(* Logix 5000 project; controller Tetris Emulate 5570 rev 35.11; software revision 35.00 *)

TASK MainTask (continuous, watchdog 500 ms) : MainProgram

MODULES
   Local : Emulate 5570 (ICP 2, rev 35.11)
END_MODULES

VAR_GLOBAL   (* controller tags *)
   AVE_Control : CONTROL := (LEN := 3);
   AVE_Dest : DINT;
   Background_Color_Matrix : SINT[12,8] := ([5,3] := 3, [6,3] := 3, [7,3] := 3, [8,3] := 3);
   Background_Matrix : SINT[12,8] := ([5,3] := 1, [6,3] := 1, [7,3] := 1, [8,3] := 1, [10,4] := 1, [10,5] := 1, [10,6] := 1, [10,7] := 1, [11,4] := 1, [11,5] := 1, [11,6] := 1, [11,7] := 1);
   Background_Saved_Color_Matrix : SINT[12,8];
   Clear_Color_Matrix : SINT[12,8];
   Clear_Matrix : SINT[12,8] := ([10,4] := 1, [10,5] := 1, [10,6] := 1, [10,7] := 1, [11,4] := 1, [11,5] := 1, [11,6] := 1, [11,7] := 1);
   Clear_Row_For_Index : DINT;
   Clock_Enable : BOOL := 1;
   CTU_Clock : COUNTER := (PRE := 2, ACC := 3, DN := 1);
   CTU_Clock_Reset : COUNTER := (PRE := 4, ACC := 3);
   Current_Piece_X_Size : DINT := 1;
   Current_Piece_Y_Size : DINT := 4;
   Current_X : SINT := 3;
   Current_Y : SINT := 5;
   Current_Y_Limit : DINT := 8;
   GSV_DateTime : DINT[7] := ([0] := 2025, [1] := 6, [2] := 5, [3] := 22, [4] := 27, [5] := 29, [6] := 833012);
   Input_Piece : SINT := 4;
   Master_Clear : BOOL;
   Next_Row_Check : SINT[8];
   ONS_Clock : BOOL := 1;
   ONS_Left : BOOL;
   ONS_Piece_Stopped : BOOL := 1;
   ONS_Right : BOOL;
   ONS_Rotate : BOOL;
   ONS_Score : BOOL[32];
   Piece_1_Matrix_R0 : SINT[2,3] := ([0,1] := 1, [1,0] := 1, [1,1] := 1, [1,2] := 1);
   Piece_1_Matrix_R1 : SINT[3,2] := ([0,0] := 1, [1,0] := 1, [1,1] := 1, [2,0] := 1);
   Piece_1_Matrix_R2 : SINT[2,3] := ([0,0] := 1, [0,1] := 1, [0,2] := 1, [1,1] := 1);
   Piece_1_Matrix_R3 : SINT[3,2] := ([0,1] := 1, [1,0] := 1, [1,1] := 1, [2,1] := 1);
   Piece_1_X : DINT;
   Piece_1_Y : INT;
   Piece_2_Matrix : SINT[2,2] := ([0,0] := 1, [0,1] := 1, [1,0] := 1, [1,1] := 1);
   Piece_3_Matrix_R0 : SINT[2,3] := ([0,0] := 1, [0,1] := 1, [1,1] := 1, [1,2] := 1);
   Piece_3_Matrix_R1 : SINT[3,2] := ([0,0] := 1, [1,0] := 1, [1,1] := 1, [2,1] := 1);
   Piece_4_Matrix_R0 : SINT[4,1] := ([0,0] := 1, [1,0] := 1, [2,0] := 1, [3,0] := 1);
   Piece_4_Matrix_R1 : SINT[1,4] := ([0,0] := 1, [0,1] := 1, [0,2] := 1, [0,3] := 1);
   Piece_Color : DINT := 3;
   Piece_Mov_Left : BOOL;
   Piece_Mov_Right : BOOL;
   Piece_Rotate : BOOL;
   Piece_Rotation : DINT;
   Piece_Type : SINT := 4;
   Previous_Color : DINT;
   Previous_Color_2 : DINT;
   Pulse_MS : BOOL;
   Reset : BOOL := 1;
   Saved_Matrix : SINT[12,8] := ([10,4] := 1, [10,5] := 1, [10,6] := 1, [10,7] := 1, [11,4] := 1, [11,5] := 1, [11,6] := 1, [11,7] := 1);
   Score : DINT;
   Start : BOOL;
   Update_Grid : BOOL;
END_VAR

PROGRAM MainProgram   (* main routine MainRoutine *)

ROUTINE Background_Clear   (* ladder *)
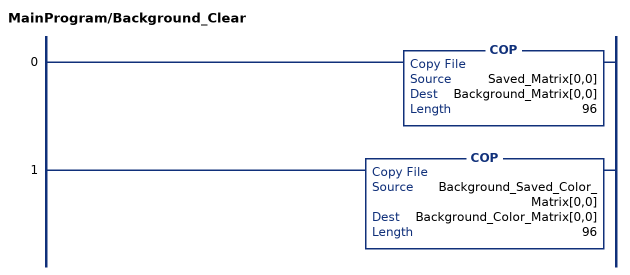
   0: COP(Saved_Matrix[0,0],Background_Matrix[0,0],96);
   1: COP(Background_Saved_Color_Matrix[0,0],Background_Color_Matrix[0,0],96);
END_ROUTINE

ROUTINE Clear_Full_Row   (* ladder *)
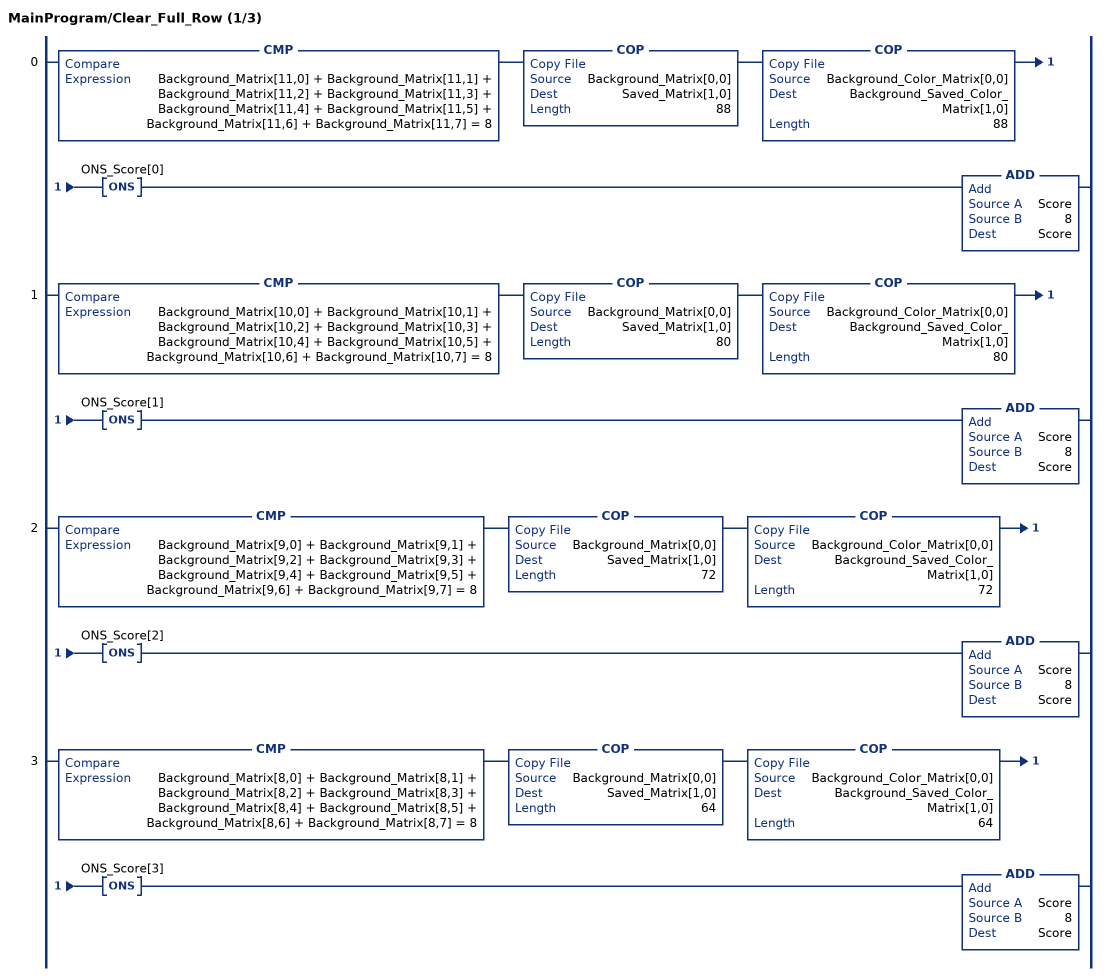
   0: CMP(Background_Matrix[11,0] + Background_Matrix[11,1] + Background_Matrix[11,2] + Background_Matrix[11,3] + Background_Matrix[11,4] + Background_Matrix[11,5] + Background_Matrix[11,6] + Background_Matrix[11,7] = 8)COP(Background_Matrix[0,0],Saved_Matrix[1,0],88)COP(Background_Color_Matrix[0,0],Background_Saved_Color_Matrix[1,0],88)ONS(ONS_Score[0])ADD(Score,8,Score);
   1: CMP(Background_Matrix[10,0] + Background_Matrix[10,1] + Background_Matrix[10,2] + Background_Matrix[10,3] + Background_Matrix[10,4] + Background_Matrix[10,5] + Background_Matrix[10,6] + Background_Matrix[10,7] = 8)COP(Background_Matrix[0,0],Saved_Matrix[1,0],80)COP(Background_Color_Matrix[0,0],Background_Saved_Color_Matrix[1,0],80)ONS(ONS_Score[1])ADD(Score,8,Score);
   2: CMP(Background_Matrix[9,0] + Background_Matrix[9,1] + Background_Matrix[9,2] + Background_Matrix[9,3] + Background_Matrix[9,4] + Background_Matrix[9,5] + Background_Matrix[9,6] + Background_Matrix[9,7] = 8)COP(Background_Matrix[0,0],Saved_Matrix[1,0],72)COP(Background_Color_Matrix[0,0],Background_Saved_Color_Matrix[1,0],72)ONS(ONS_Score[2])ADD(Score,8,Score);
   3: CMP(Background_Matrix[8,0] + Background_Matrix[8,1] + Background_Matrix[8,2] + Background_Matrix[8,3] + Background_Matrix[8,4] + Background_Matrix[8,5] + Background_Matrix[8,6] + Background_Matrix[8,7] = 8)COP(Background_Matrix[0,0],Saved_Matrix[1,0],64)COP(Background_Color_Matrix[0,0],Background_Saved_Color_Matrix[1,0],64)ONS(ONS_Score[3])ADD(Score,8,Score);
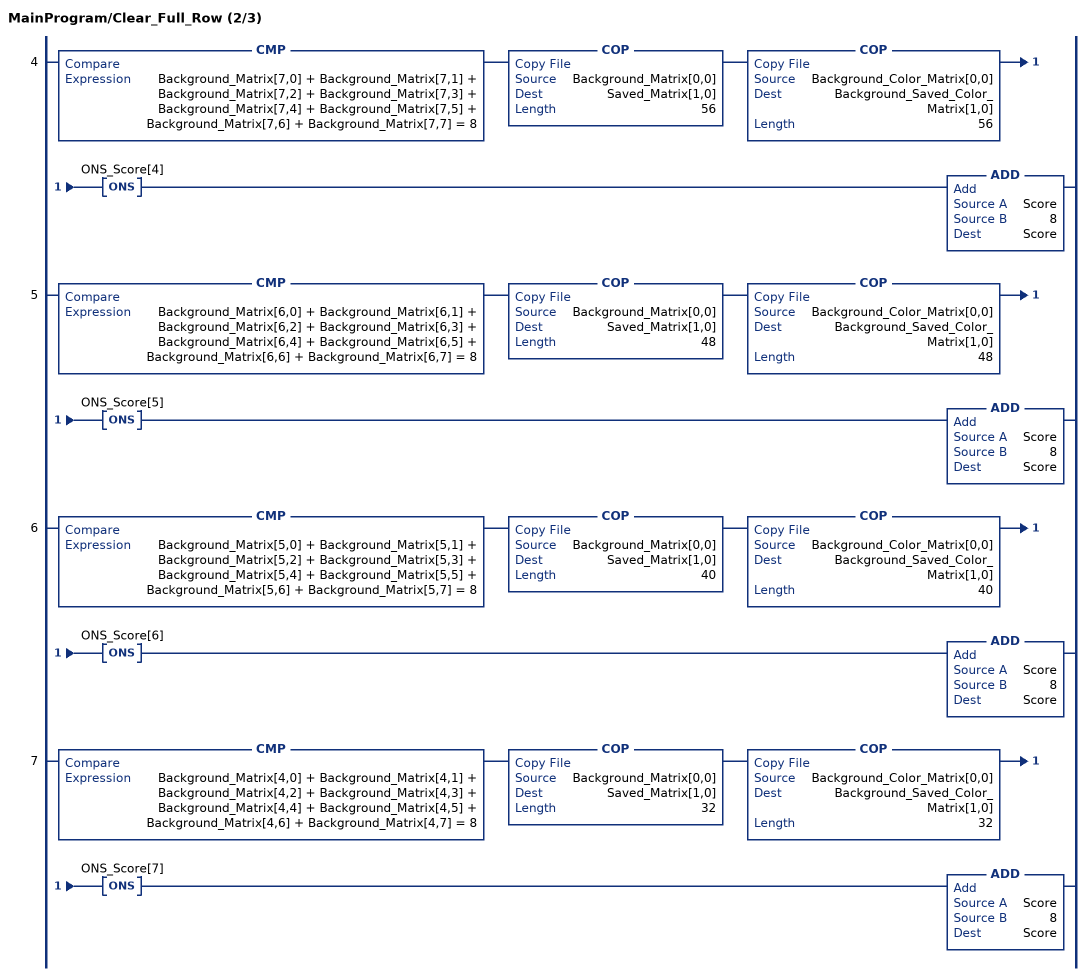
   4: CMP(Background_Matrix[7,0] + Background_Matrix[7,1] + Background_Matrix[7,2] + Background_Matrix[7,3] + Background_Matrix[7,4] + Background_Matrix[7,5] + Background_Matrix[7,6] + Background_Matrix[7,7] = 8)COP(Background_Matrix[0,0],Saved_Matrix[1,0],56)COP(Background_Color_Matrix[0,0],Background_Saved_Color_Matrix[1,0],56)ONS(ONS_Score[4])ADD(Score,8,Score);
   5: CMP(Background_Matrix[6,0] + Background_Matrix[6,1] + Background_Matrix[6,2] + Background_Matrix[6,3] + Background_Matrix[6,4] + Background_Matrix[6,5] + Background_Matrix[6,6] + Background_Matrix[6,7] = 8)COP(Background_Matrix[0,0],Saved_Matrix[1,0],48)COP(Background_Color_Matrix[0,0],Background_Saved_Color_Matrix[1,0],48)ONS(ONS_Score[5])ADD(Score,8,Score);
   6: CMP(Background_Matrix[5,0] + Background_Matrix[5,1] + Background_Matrix[5,2] + Background_Matrix[5,3] + Background_Matrix[5,4] + Background_Matrix[5,5] + Background_Matrix[5,6] + Background_Matrix[5,7] = 8)COP(Background_Matrix[0,0],Saved_Matrix[1,0],40)COP(Background_Color_Matrix[0,0],Background_Saved_Color_Matrix[1,0],40)ONS(ONS_Score[6])ADD(Score,8,Score);
   7: CMP(Background_Matrix[4,0] + Background_Matrix[4,1] + Background_Matrix[4,2] + Background_Matrix[4,3] + Background_Matrix[4,4] + Background_Matrix[4,5] + Background_Matrix[4,6] + Background_Matrix[4,7] = 8)COP(Background_Matrix[0,0],Saved_Matrix[1,0],32)COP(Background_Color_Matrix[0,0],Background_Saved_Color_Matrix[1,0],32)ONS(ONS_Score[7])ADD(Score,8,Score);
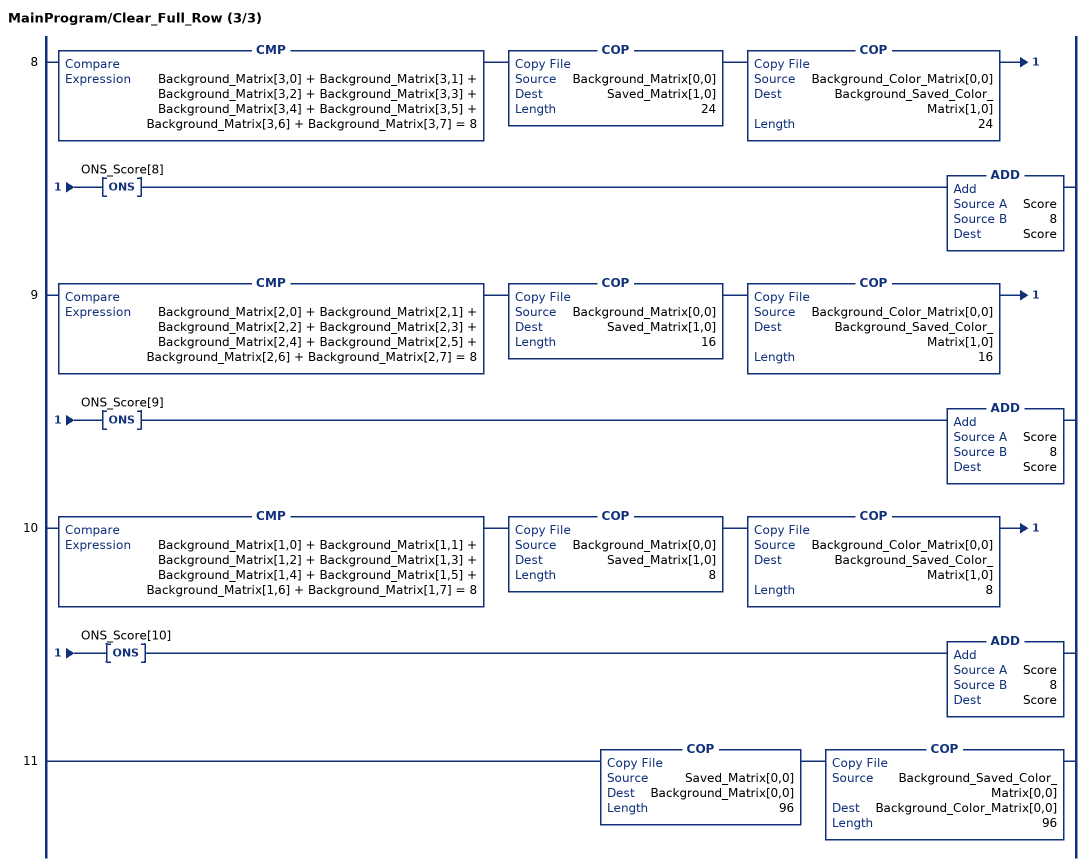
   8: CMP(Background_Matrix[3,0] + Background_Matrix[3,1] + Background_Matrix[3,2] + Background_Matrix[3,3] + Background_Matrix[3,4] + Background_Matrix[3,5] + Background_Matrix[3,6] + Background_Matrix[3,7] = 8)COP(Background_Matrix[0,0],Saved_Matrix[1,0],24)COP(Background_Color_Matrix[0,0],Background_Saved_Color_Matrix[1,0],24)ONS(ONS_Score[8])ADD(Score,8,Score);
   9: CMP(Background_Matrix[2,0] + Background_Matrix[2,1] + Background_Matrix[2,2] + Background_Matrix[2,3] + Background_Matrix[2,4] + Background_Matrix[2,5] + Background_Matrix[2,6] + Background_Matrix[2,7] = 8)COP(Background_Matrix[0,0],Saved_Matrix[1,0],16)COP(Background_Color_Matrix[0,0],Background_Saved_Color_Matrix[1,0],16)ONS(ONS_Score[9])ADD(Score,8,Score);
   10: CMP(Background_Matrix[1,0] + Background_Matrix[1,1] + Background_Matrix[1,2] + Background_Matrix[1,3] + Background_Matrix[1,4] + Background_Matrix[1,5] + Background_Matrix[1,6] + Background_Matrix[1,7] = 8)COP(Background_Matrix[0,0],Saved_Matrix[1,0],8)COP(Background_Color_Matrix[0,0],Background_Saved_Color_Matrix[1,0],8)ONS(ONS_Score[10])ADD(Score,8,Score);
   11: COP(Saved_Matrix[0,0],Background_Matrix[0,0],96)COP(Background_Saved_Color_Matrix[0,0],Background_Color_Matrix[0,0],96);
END_ROUTINE

ROUTINE Clock   (* ladder *)
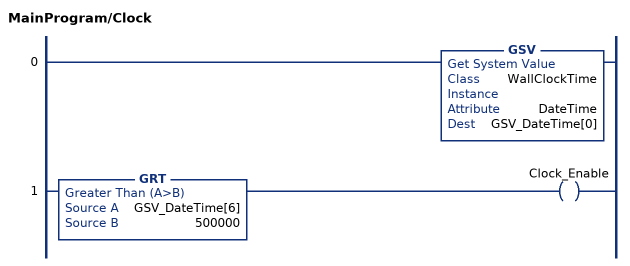
   0: GSV(WallClockTime,,DateTime,GSV_DateTime[0]);
   1: GRT(GSV_DateTime[6],500000)OTE(Clock_Enable);
END_ROUTINE

ROUTINE MainRoutine   (* ladder *)
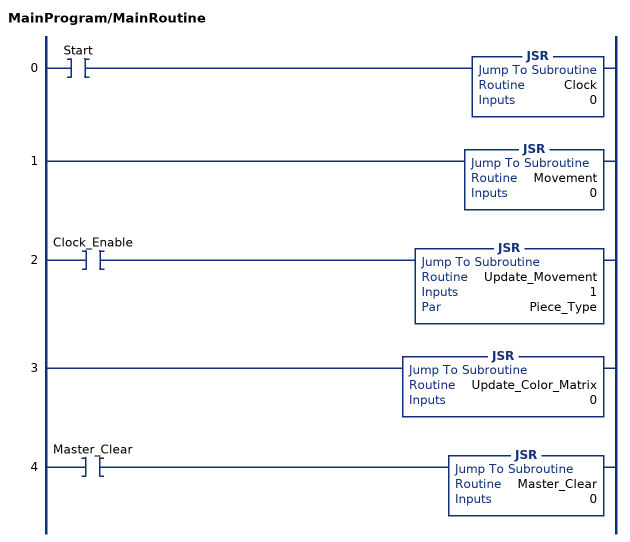
   0: XIC(Start)JSR(Clock,0);
   1: JSR(Movement,0);
   2: XIC(Clock_Enable)JSR(Update_Movement,1,Piece_Type);
   3: JSR(Update_Color_Matrix,0);
   4: XIC(Master_Clear)JSR(Master_Clear,0);
END_ROUTINE

ROUTINE Master_Clear   (* ladder *)
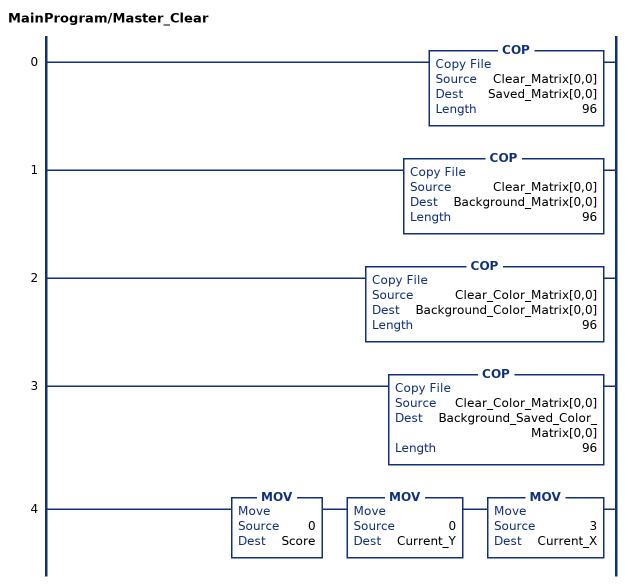
   0: COP(Clear_Matrix[0,0],Saved_Matrix[0,0],96);
   1: COP(Clear_Matrix[0,0],Background_Matrix[0,0],96);
   2: COP(Clear_Color_Matrix[0,0],Background_Color_Matrix[0,0],96);
   3: COP(Clear_Color_Matrix[0,0],Background_Saved_Color_Matrix[0,0],96);
   4: MOV(0,Score)MOV(0,Current_Y)MOV(3,Current_X);
END_ROUTINE

ROUTINE Movement   (* ladder *)
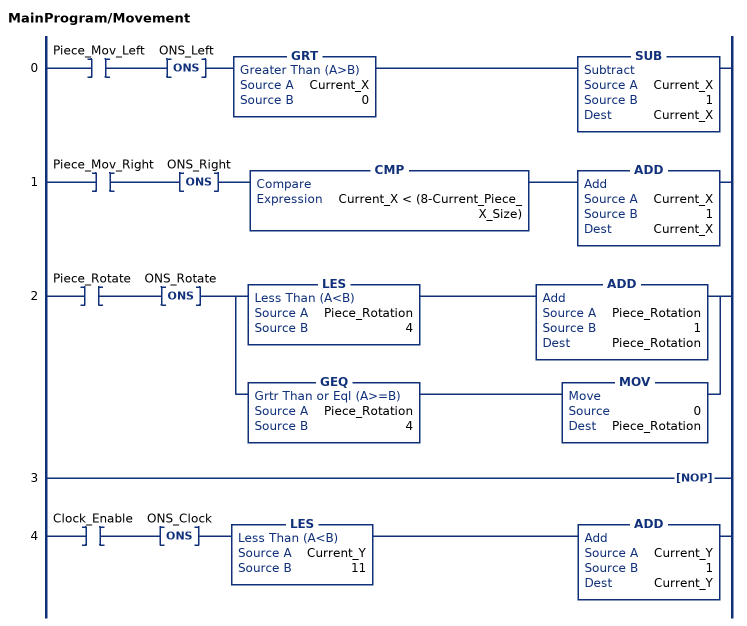
   0: XIC(Piece_Mov_Left)ONS(ONS_Left)GRT(Current_X,0)SUB(Current_X,1,Current_X);
   1: XIC(Piece_Mov_Right)ONS(ONS_Right)CMP(Current_X < (8-Current_Piece_X_Size))ADD(Current_X,1,Current_X);
   2: XIC(Piece_Rotate)ONS(ONS_Rotate)[LES(Piece_Rotation,4) ADD(Piece_Rotation,1,Piece_Rotation) ,GEQ(Piece_Rotation,4) MOV(0,Piece_Rotation) ];
   3: NOP();
   4: XIC(Clock_Enable)ONS(ONS_Clock)LES(Current_Y,11)ADD(Current_Y,1,Current_Y);
END_ROUTINE

ROUTINE Piece_1_Rotation   (* ladder *)
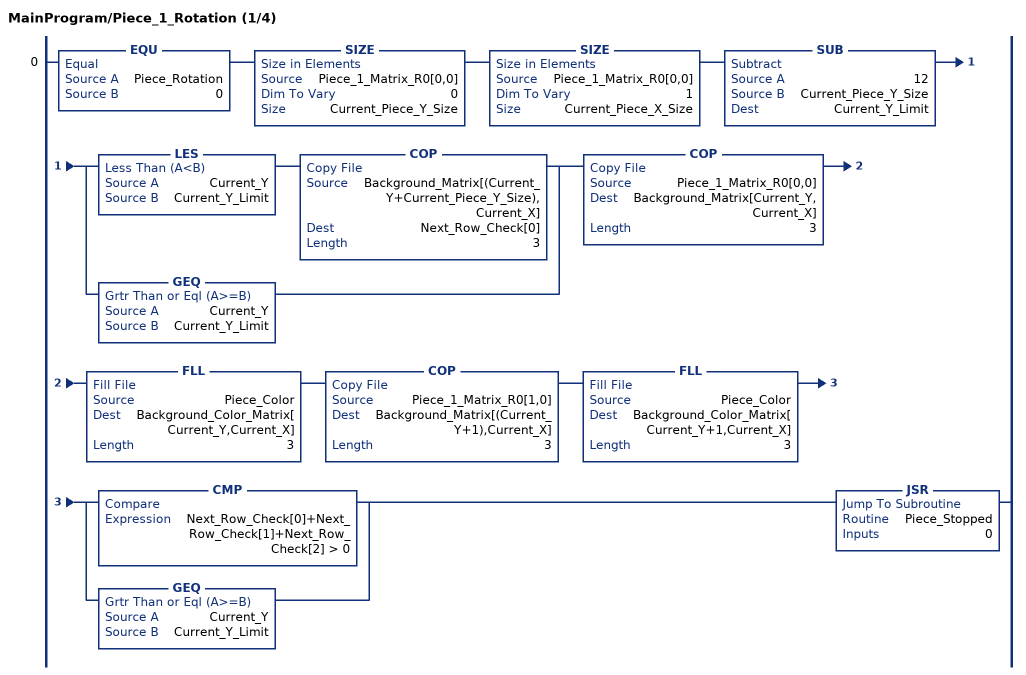
   0: EQU(Piece_Rotation,0)SIZE(Piece_1_Matrix_R0[0,0],0,Current_Piece_Y_Size)SIZE(Piece_1_Matrix_R0[0,0],1,Current_Piece_X_Size)SUB(12,Current_Piece_Y_Size,Current_Y_Limit)[LES(Current_Y,Current_Y_Limit) COP(Background_Matrix[(Current_Y+Current_Piece_Y_Size),Current_X],Next_Row_Check[0],3) ,GEQ(Current_Y,Current_Y_Limit) ]COP(Piece_1_Matrix_R0[0,0],Background_Matrix[Current_Y,Current_X],3)FLL(Piece_Color,Background_Color_Matrix[Current_Y,Current_X],3)COP(Piece_1_Matrix_R0[1,0],Background_Matrix[(Current_Y+1),Current_X],3)FLL(Piece_Color,Background_Color_Matrix[Current_Y+1,Current_X],3)[CMP(Next_Row_Check[0]+Next_Row_Check[1]+Next_Row_Check[2] > 0) ,GEQ(Current_Y,Current_Y_Limit) ]JSR(Piece_Stopped,0);
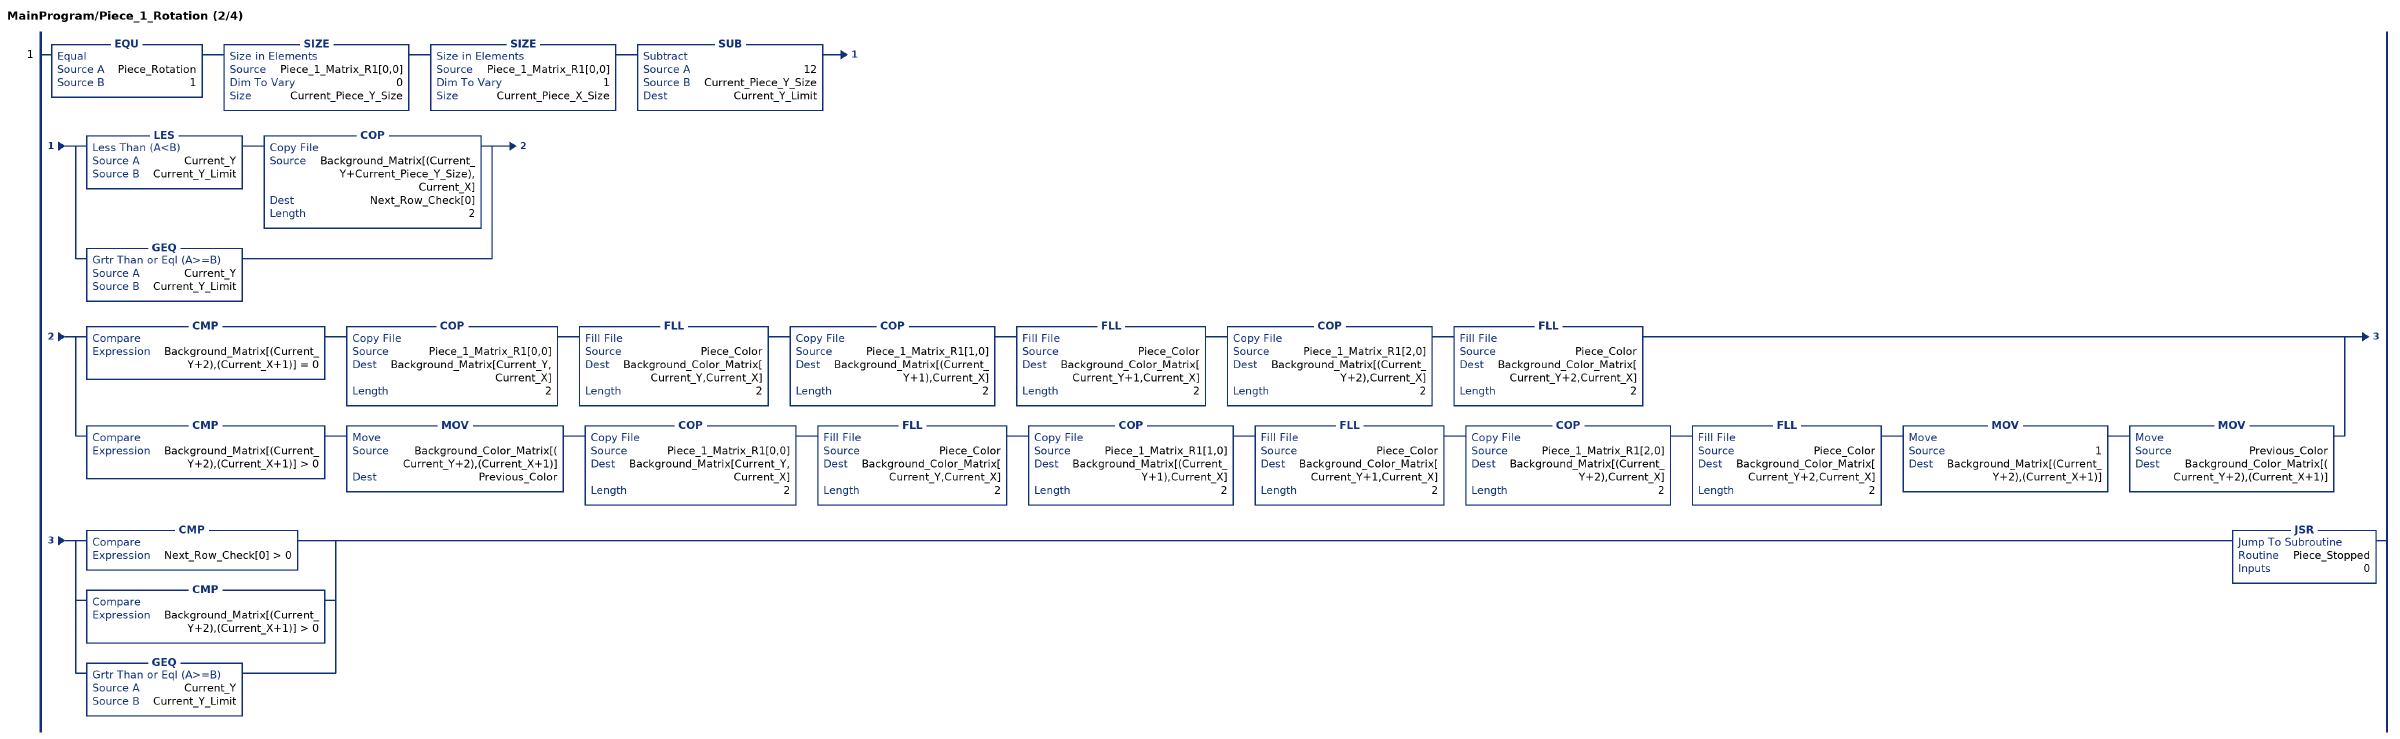
   1: EQU(Piece_Rotation,1)SIZE(Piece_1_Matrix_R1[0,0],0,Current_Piece_Y_Size)SIZE(Piece_1_Matrix_R1[0,0],1,Current_Piece_X_Size)SUB(12,Current_Piece_Y_Size,Current_Y_Limit)[LES(Current_Y,Current_Y_Limit) COP(Background_Matrix[(Current_Y+Current_Piece_Y_Size),Current_X],Next_Row_Check[0],2) ,GEQ(Current_Y,Current_Y_Limit) ][CMP(Background_Matrix[(Current_Y+2),(Current_X+1)] = 0) COP(Piece_1_Matrix_R1[0,0],Background_Matrix[Current_Y,Current_X],2) FLL(Piece_Color,Background_Color_Matrix[Current_Y,Current_X],2) COP(Piece_1_Matrix_R1[1,0],Background_Matrix[(Current_Y+1),Current_X],2) FLL(Piece_Color,Background_Color_Matrix[Current_Y+1,Current_X],2) COP(Piece_1_Matrix_R1[2,0],Background_Matrix[(Current_Y+2),Current_X],2) FLL(Piece_Color,Background_Color_Matrix[Current_Y+2,Current_X],2) ,CMP(Background_Matrix[(Current_Y+2),(Current_X+1)] > 0) MOV(Background_Color_Matrix[(Current_Y+2),(Current_X+1)],Previous_Color) COP(Piece_1_Matrix_R1[0,0],Background_Matrix[Current_Y,Current_X],2) FLL(Piece_Color,Background_Color_Matrix[Current_Y,Current_X],2) COP(Piece_1_Matrix_R1[1,0],Background_Matrix[(Current_Y+1),Current_X],2) FLL(Piece_Color,Background_Color_Matrix[Current_Y+1,Current_X],2) COP(Piece_1_Matrix_R1[2,0],Background_Matrix[(Current_Y+2),Current_X],2) FLL(Piece_Color,Background_Color_Matrix[Current_Y+2,Current_X],2) MOV(1,Background_Matrix[(Current_Y+2),(Current_X+1)]) MOV(Previous_Color,Background_Color_Matrix[(Current_Y+2),(Current_X+1)]) ][CMP(Next_Row_Check[0] > 0) ,CMP(Background_Matrix[(Current_Y+2),(Current_X+1)] > 0) ,GEQ(Current_Y,Current_Y_Limit) ]JSR(Piece_Stopped,0);
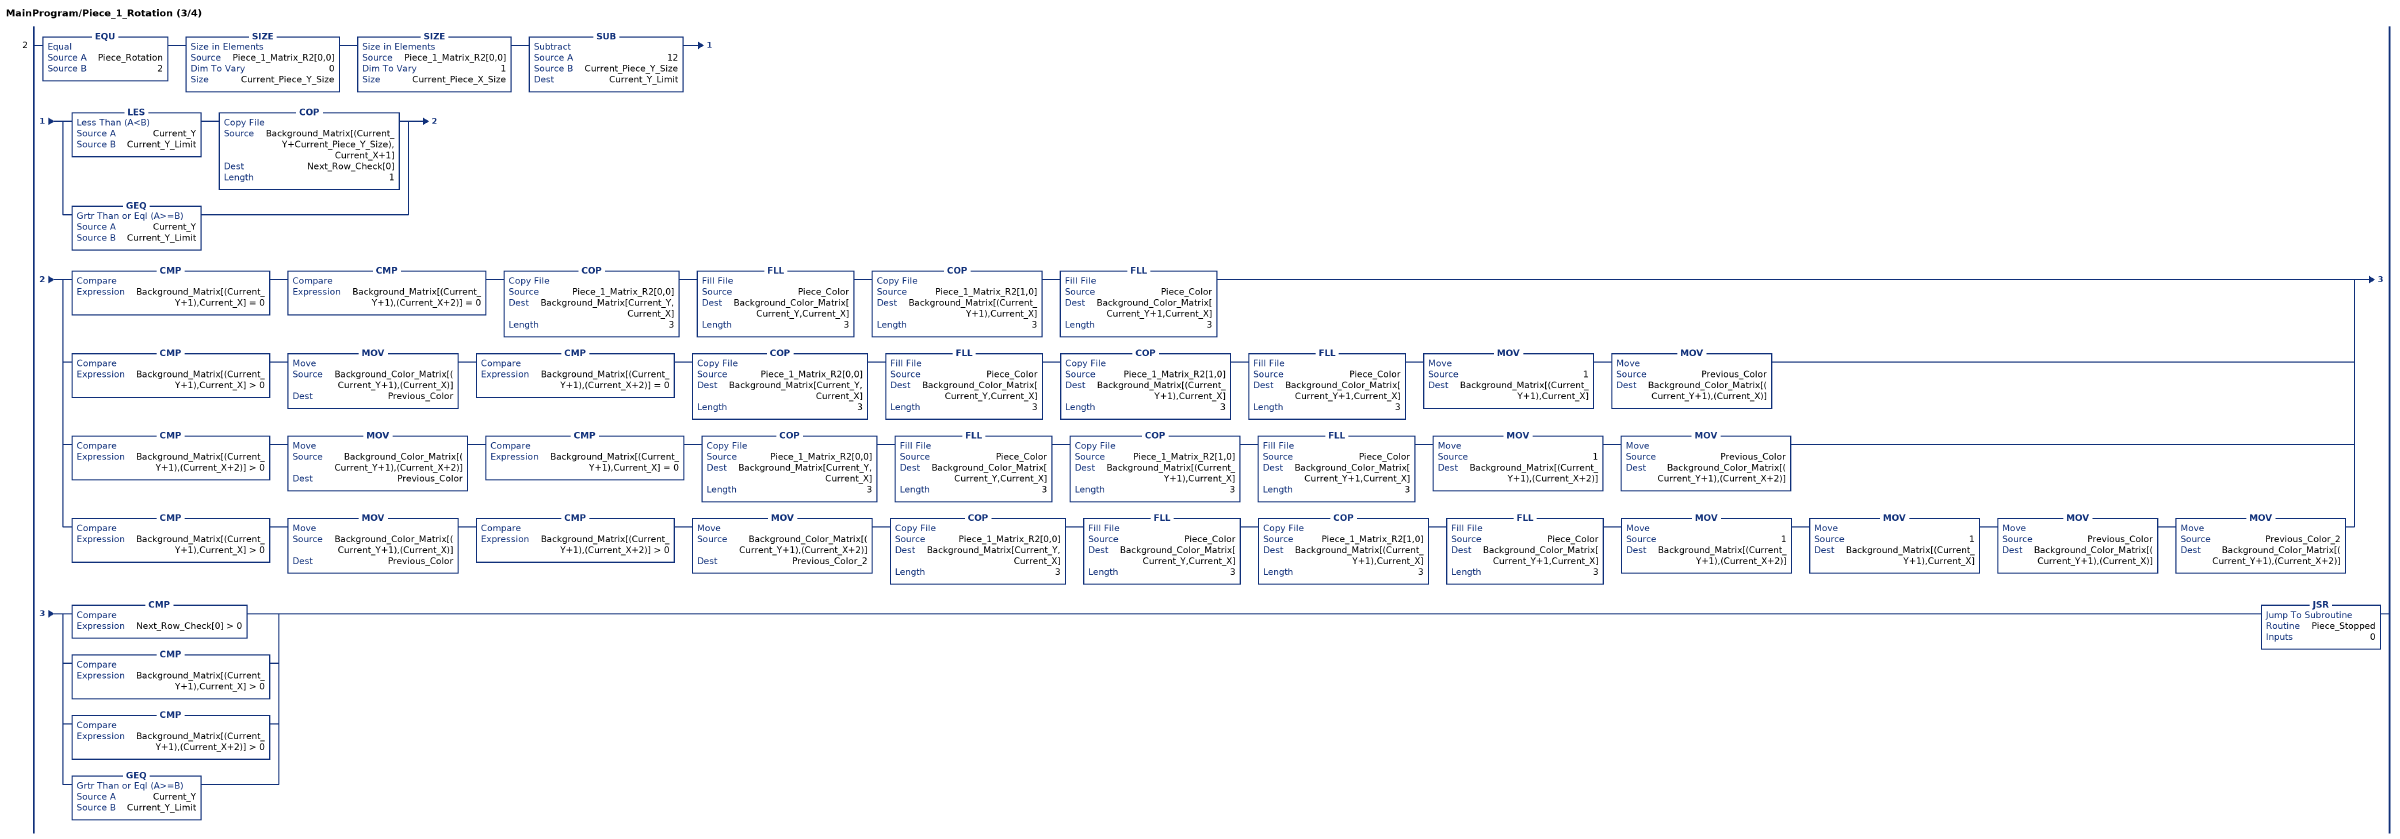
   2: EQU(Piece_Rotation,2)SIZE(Piece_1_Matrix_R2[0,0],0,Current_Piece_Y_Size)SIZE(Piece_1_Matrix_R2[0,0],1,Current_Piece_X_Size)SUB(12,Current_Piece_Y_Size,Current_Y_Limit)[LES(Current_Y,Current_Y_Limit) COP(Background_Matrix[(Current_Y+Current_Piece_Y_Size),Current_X+1],Next_Row_Check[0],1) ,GEQ(Current_Y,Current_Y_Limit) ][CMP(Background_Matrix[(Current_Y+1),Current_X] = 0) CMP(Background_Matrix[(Current_Y+1),(Current_X+2)] = 0) COP(Piece_1_Matrix_R2[0,0],Background_Matrix[Current_Y,Current_X],3) FLL(Piece_Color,Background_Color_Matrix[Current_Y,Current_X],3) COP(Piece_1_Matrix_R2[1,0],Background_Matrix[(Current_Y+1),Current_X],3) FLL(Piece_Color,Background_Color_Matrix[Current_Y+1,Current_X],3) ,[CMP(Background_Matrix[(Current_Y+1),Current_X] > 0) MOV(Background_Color_Matrix[(Current_Y+1),(Current_X)],Previous_Color) CMP(Background_Matrix[(Current_Y+1),(Current_X+2)] = 0) COP(Piece_1_Matrix_R2[0,0],Background_Matrix[Current_Y,Current_X],3) FLL(Piece_Color,Background_Color_Matrix[Current_Y,Current_X],3) COP(Piece_1_Matrix_R2[1,0],Background_Matrix[(Current_Y+1),Current_X],3) FLL(Piece_Color,Background_Color_Matrix[Current_Y+1,Current_X],3) MOV(1,Background_Matrix[(Current_Y+1),Current_X]) MOV(Previous_Color,Background_Color_Matrix[(Current_Y+1),(Current_X)]) ,[CMP(Background_Matrix[(Current_Y+1),(Current_X+2)] > 0) MOV(Background_Color_Matrix[(Current_Y+1),(Current_X+2)],Previous_Color) CMP(Background_Matrix[(Current_Y+1),Current_X] = 0) COP(Piece_1_Matrix_R2[0,0],Background_Matrix[Current_Y,Current_X],3) FLL(Piece_Color,Background_Color_Matrix[Current_Y,Current_X],3) COP(Piece_1_Matrix_R2[1,0],Background_Matrix[(Current_Y+1),Current_X],3) FLL(Piece_Color,Background_Color_Matrix[Current_Y+1,Current_X],3) MOV(1,Background_Matrix[(Current_Y+1),(Current_X+2)]) MOV(Previous_Color,Background_Color_Matrix[(Current_Y+1),(Current_X+2)]) ,CMP(Background_Matrix[(Current_Y+1),Current_X] > 0) MOV(Background_Color_Matrix[(Current_Y+1),(Current_X)],Previous_Color) CMP(Background_Matrix[(Current_Y+1),(Current_X+2)] > 0) MOV(Background_Color_Matrix[(Current_Y+1),(Current_X+2)],Previous_Color_2) COP(Piece_1_Matrix_R2[0,0],Background_Matrix[Current_Y,Current_X],3) FLL(Piece_Color,Background_Color_Matrix[Current_Y,Current_X],3) COP(Piece_1_Matrix_R2[1,0],Background_Matrix[(Current_Y+1),Current_X],3) FLL(Piece_Color,Background_Color_Matrix[Current_Y+1,Current_X],3) MOV(1,Background_Matrix[(Current_Y+1),(Current_X+2)]) MOV(1,Background_Matrix[(Current_Y+1),Current_X]) MOV(Previous_Color,Background_Color_Matrix[(Current_Y+1),(Current_X)]) MOV(Previous_Color_2,Background_Color_Matrix[(Current_Y+1),(Current_X+2)]) ] ] ][CMP(Next_Row_Check[0] > 0) ,CMP(Background_Matrix[(Current_Y+1),Current_X] > 0) ,CMP(Background_Matrix[(Current_Y+1),(Current_X+2)] > 0) ,GEQ(Current_Y,Current_Y_Limit) ]JSR(Piece_Stopped,0);
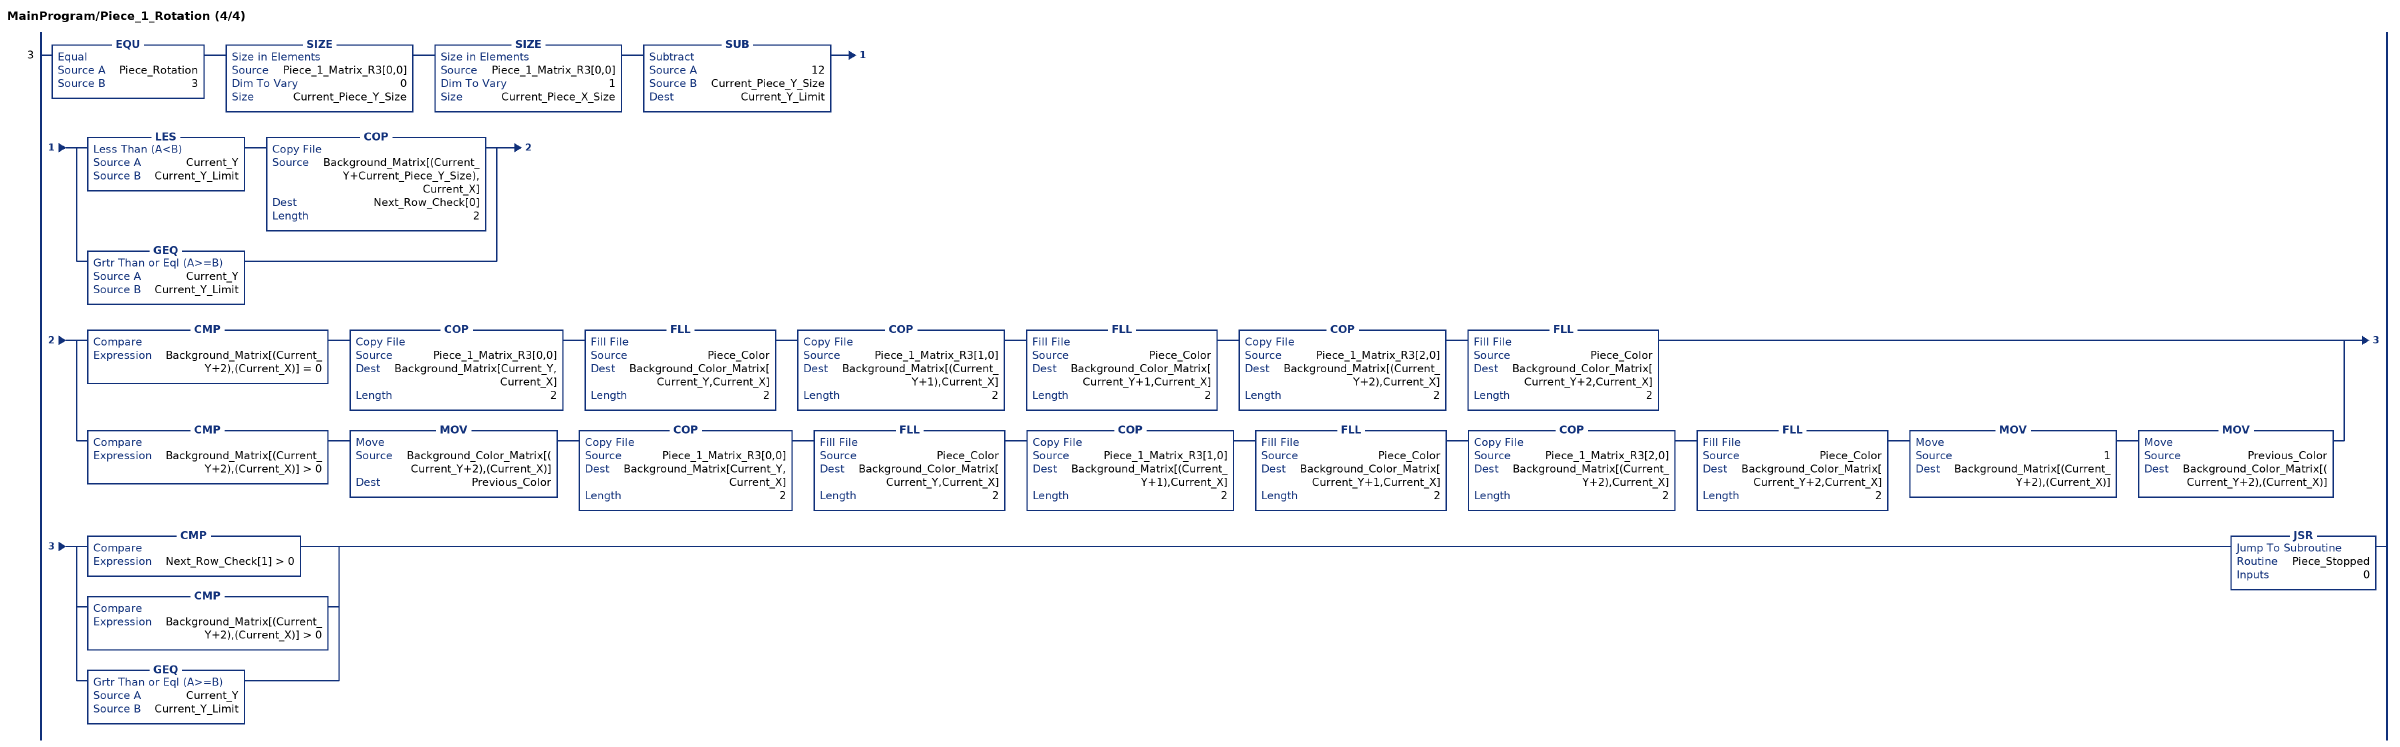
   3: EQU(Piece_Rotation,3)SIZE(Piece_1_Matrix_R3[0,0],0,Current_Piece_Y_Size)SIZE(Piece_1_Matrix_R3[0,0],1,Current_Piece_X_Size)SUB(12,Current_Piece_Y_Size,Current_Y_Limit)[LES(Current_Y,Current_Y_Limit) COP(Background_Matrix[(Current_Y+Current_Piece_Y_Size),Current_X],Next_Row_Check[0],2) ,GEQ(Current_Y,Current_Y_Limit) ][CMP(Background_Matrix[(Current_Y+2),(Current_X)] = 0) COP(Piece_1_Matrix_R3[0,0],Background_Matrix[Current_Y,Current_X],2) FLL(Piece_Color,Background_Color_Matrix[Current_Y,Current_X],2) COP(Piece_1_Matrix_R3[1,0],Background_Matrix[(Current_Y+1),Current_X],2) FLL(Piece_Color,Background_Color_Matrix[Current_Y+1,Current_X],2) COP(Piece_1_Matrix_R3[2,0],Background_Matrix[(Current_Y+2),Current_X],2) FLL(Piece_Color,Background_Color_Matrix[Current_Y+2,Current_X],2) ,CMP(Background_Matrix[(Current_Y+2),(Current_X)] > 0) MOV(Background_Color_Matrix[(Current_Y+2),(Current_X)],Previous_Color) COP(Piece_1_Matrix_R3[0,0],Background_Matrix[Current_Y,Current_X],2) FLL(Piece_Color,Background_Color_Matrix[Current_Y,Current_X],2) COP(Piece_1_Matrix_R3[1,0],Background_Matrix[(Current_Y+1),Current_X],2) FLL(Piece_Color,Background_Color_Matrix[Current_Y+1,Current_X],2) COP(Piece_1_Matrix_R3[2,0],Background_Matrix[(Current_Y+2),Current_X],2) FLL(Piece_Color,Background_Color_Matrix[Current_Y+2,Current_X],2) MOV(1,Background_Matrix[(Current_Y+2),(Current_X)]) MOV(Previous_Color,Background_Color_Matrix[(Current_Y+2),(Current_X)]) ][CMP(Next_Row_Check[1] > 0) ,CMP(Background_Matrix[(Current_Y+2),(Current_X)] > 0) ,GEQ(Current_Y,Current_Y_Limit) ]JSR(Piece_Stopped,0);
END_ROUTINE

ROUTINE Piece_3_Rotation   (* ladder *)
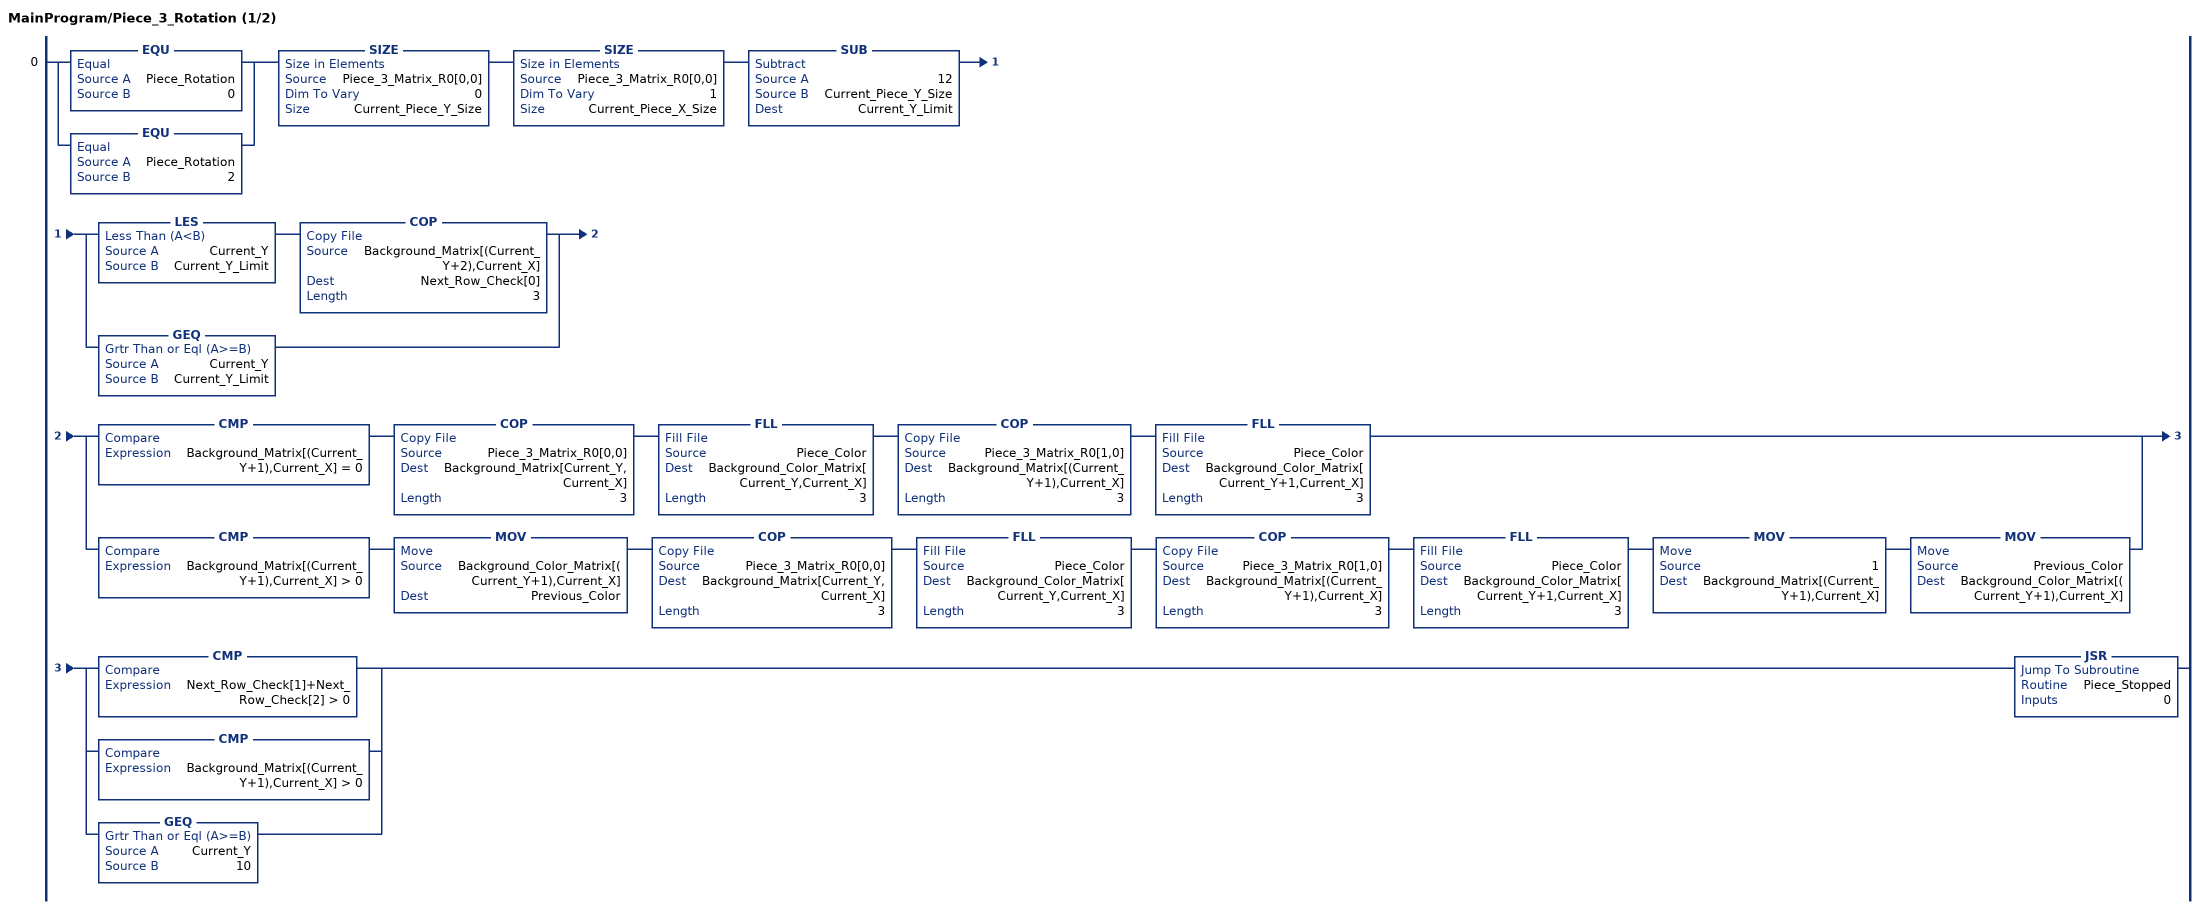
   0: [EQU(Piece_Rotation,0) ,EQU(Piece_Rotation,2) ]SIZE(Piece_3_Matrix_R0[0,0],0,Current_Piece_Y_Size)SIZE(Piece_3_Matrix_R0[0,0],1,Current_Piece_X_Size)SUB(12,Current_Piece_Y_Size,Current_Y_Limit)[LES(Current_Y,Current_Y_Limit) COP(Background_Matrix[(Current_Y+2),Current_X],Next_Row_Check[0],3) ,GEQ(Current_Y,Current_Y_Limit) ][CMP(Background_Matrix[(Current_Y+1),Current_X] = 0) COP(Piece_3_Matrix_R0[0,0],Background_Matrix[Current_Y,Current_X],3) FLL(Piece_Color,Background_Color_Matrix[Current_Y,Current_X],3) COP(Piece_3_Matrix_R0[1,0],Background_Matrix[(Current_Y+1),Current_X],3) FLL(Piece_Color,Background_Color_Matrix[Current_Y+1,Current_X],3) ,CMP(Background_Matrix[(Current_Y+1),Current_X] > 0) MOV(Background_Color_Matrix[(Current_Y+1),Current_X],Previous_Color) COP(Piece_3_Matrix_R0[0,0],Background_Matrix[Current_Y,Current_X],3) FLL(Piece_Color,Background_Color_Matrix[Current_Y,Current_X],3) COP(Piece_3_Matrix_R0[1,0],Background_Matrix[(Current_Y+1),Current_X],3) FLL(Piece_Color,Background_Color_Matrix[Current_Y+1,Current_X],3) MOV(1,Background_Matrix[(Current_Y+1),Current_X]) MOV(Previous_Color,Background_Color_Matrix[(Current_Y+1),Current_X]) ][CMP(Next_Row_Check[1]+Next_Row_Check[2] > 0) ,CMP(Background_Matrix[(Current_Y+1),Current_X] > 0) ,GEQ(Current_Y,10) ]JSR(Piece_Stopped,0);
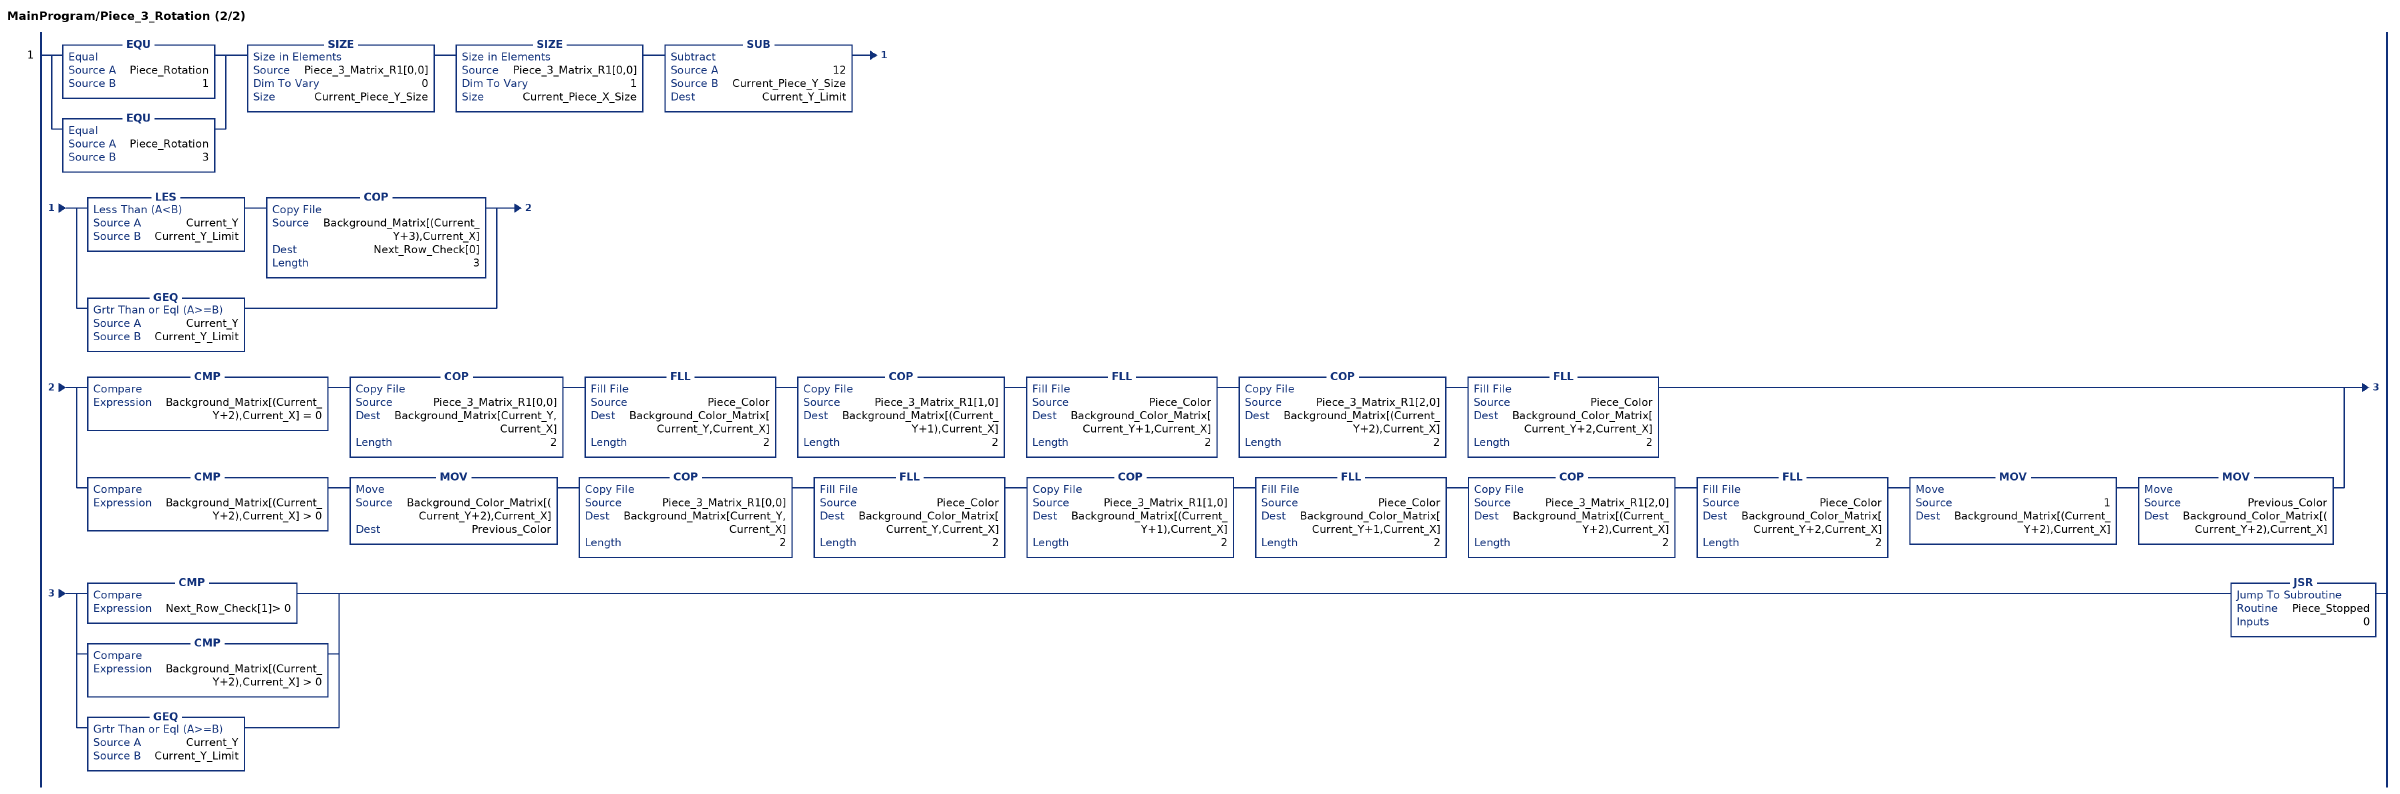
   1: [EQU(Piece_Rotation,1) ,EQU(Piece_Rotation,3) ]SIZE(Piece_3_Matrix_R1[0,0],0,Current_Piece_Y_Size)SIZE(Piece_3_Matrix_R1[0,0],1,Current_Piece_X_Size)SUB(12,Current_Piece_Y_Size,Current_Y_Limit)[LES(Current_Y,Current_Y_Limit) COP(Background_Matrix[(Current_Y+3),Current_X],Next_Row_Check[0],3) ,GEQ(Current_Y,Current_Y_Limit) ][CMP(Background_Matrix[(Current_Y+2),Current_X] = 0) COP(Piece_3_Matrix_R1[0,0],Background_Matrix[Current_Y,Current_X],2) FLL(Piece_Color,Background_Color_Matrix[Current_Y,Current_X],2) COP(Piece_3_Matrix_R1[1,0],Background_Matrix[(Current_Y+1),Current_X],2) FLL(Piece_Color,Background_Color_Matrix[Current_Y+1,Current_X],2) COP(Piece_3_Matrix_R1[2,0],Background_Matrix[(Current_Y+2),Current_X],2) FLL(Piece_Color,Background_Color_Matrix[Current_Y+2,Current_X],2) ,CMP(Background_Matrix[(Current_Y+2),Current_X] > 0) MOV(Background_Color_Matrix[(Current_Y+2),Current_X],Previous_Color) COP(Piece_3_Matrix_R1[0,0],Background_Matrix[Current_Y,Current_X],2) FLL(Piece_Color,Background_Color_Matrix[Current_Y,Current_X],2) COP(Piece_3_Matrix_R1[1,0],Background_Matrix[(Current_Y+1),Current_X],2) FLL(Piece_Color,Background_Color_Matrix[Current_Y+1,Current_X],2) COP(Piece_3_Matrix_R1[2,0],Background_Matrix[(Current_Y+2),Current_X],2) FLL(Piece_Color,Background_Color_Matrix[Current_Y+2,Current_X],2) MOV(1,Background_Matrix[(Current_Y+2),Current_X]) MOV(Previous_Color,Background_Color_Matrix[(Current_Y+2),Current_X]) ][CMP(Next_Row_Check[1]> 0) ,CMP(Background_Matrix[(Current_Y+2),Current_X] > 0) ,GEQ(Current_Y,Current_Y_Limit) ]JSR(Piece_Stopped,0);
END_ROUTINE

ROUTINE Piece_4_Rotation   (* ladder *)
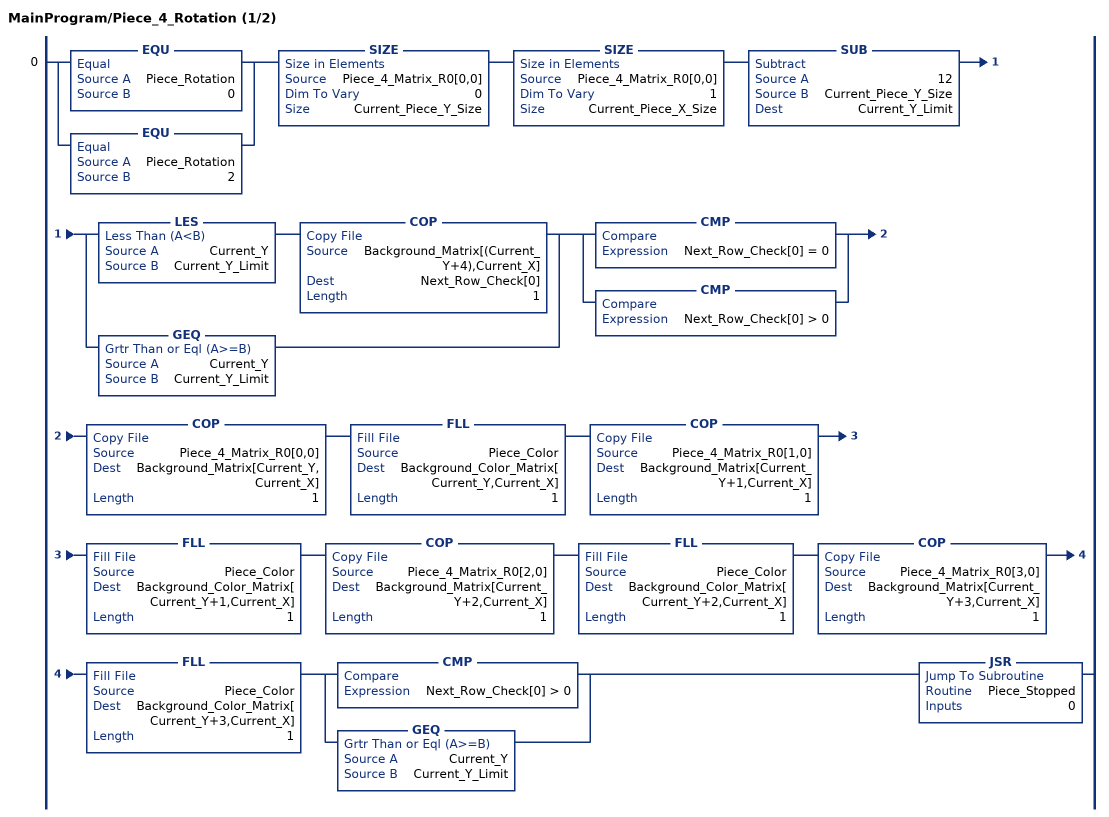
   0: [EQU(Piece_Rotation,0) ,EQU(Piece_Rotation,2) ]SIZE(Piece_4_Matrix_R0[0,0],0,Current_Piece_Y_Size)SIZE(Piece_4_Matrix_R0[0,0],1,Current_Piece_X_Size)SUB(12,Current_Piece_Y_Size,Current_Y_Limit)[LES(Current_Y,Current_Y_Limit) COP(Background_Matrix[(Current_Y+4),Current_X],Next_Row_Check[0],1) ,GEQ(Current_Y,Current_Y_Limit) ][CMP(Next_Row_Check[0] = 0) ,CMP(Next_Row_Check[0] > 0) ]COP(Piece_4_Matrix_R0[0,0],Background_Matrix[Current_Y,Current_X],1)FLL(Piece_Color,Background_Color_Matrix[Current_Y,Current_X],1)COP(Piece_4_Matrix_R0[1,0],Background_Matrix[Current_Y+1,Current_X],1)FLL(Piece_Color,Background_Color_Matrix[Current_Y+1,Current_X],1)COP(Piece_4_Matrix_R0[2,0],Background_Matrix[Current_Y+2,Current_X],1)FLL(Piece_Color,Background_Color_Matrix[Current_Y+2,Current_X],1)COP(Piece_4_Matrix_R0[3,0],Background_Matrix[Current_Y+3,Current_X],1)FLL(Piece_Color,Background_Color_Matrix[Current_Y+3,Current_X],1)[CMP(Next_Row_Check[0] > 0) ,GEQ(Current_Y,Current_Y_Limit) ]JSR(Piece_Stopped,0);
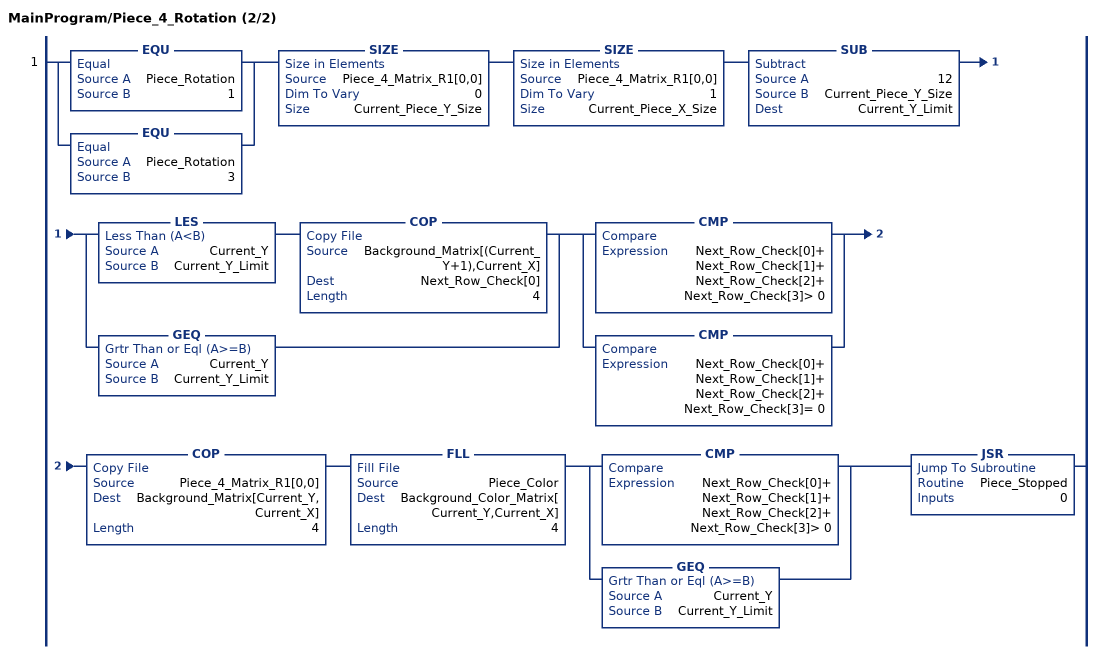
   1: [EQU(Piece_Rotation,1) ,EQU(Piece_Rotation,3) ]SIZE(Piece_4_Matrix_R1[0,0],0,Current_Piece_Y_Size)SIZE(Piece_4_Matrix_R1[0,0],1,Current_Piece_X_Size)SUB(12,Current_Piece_Y_Size,Current_Y_Limit)[LES(Current_Y,Current_Y_Limit) COP(Background_Matrix[(Current_Y+1),Current_X],Next_Row_Check[0],4) ,GEQ(Current_Y,Current_Y_Limit) ][CMP(Next_Row_Check[0]+ Next_Row_Check[1]+ Next_Row_Check[2]+ Next_Row_Check[3]> 0) ,CMP(Next_Row_Check[0]+ Next_Row_Check[1]+ Next_Row_Check[2]+ Next_Row_Check[3]= 0) ]COP(Piece_4_Matrix_R1[0,0],Background_Matrix[Current_Y,Current_X],4)FLL(Piece_Color,Background_Color_Matrix[Current_Y,Current_X],4)[CMP(Next_Row_Check[0]+ Next_Row_Check[1]+ Next_Row_Check[2]+ Next_Row_Check[3]> 0) ,GEQ(Current_Y,Current_Y_Limit) ]JSR(Piece_Stopped,0);
END_ROUTINE

ROUTINE Piece_Stopped   (* ladder *)
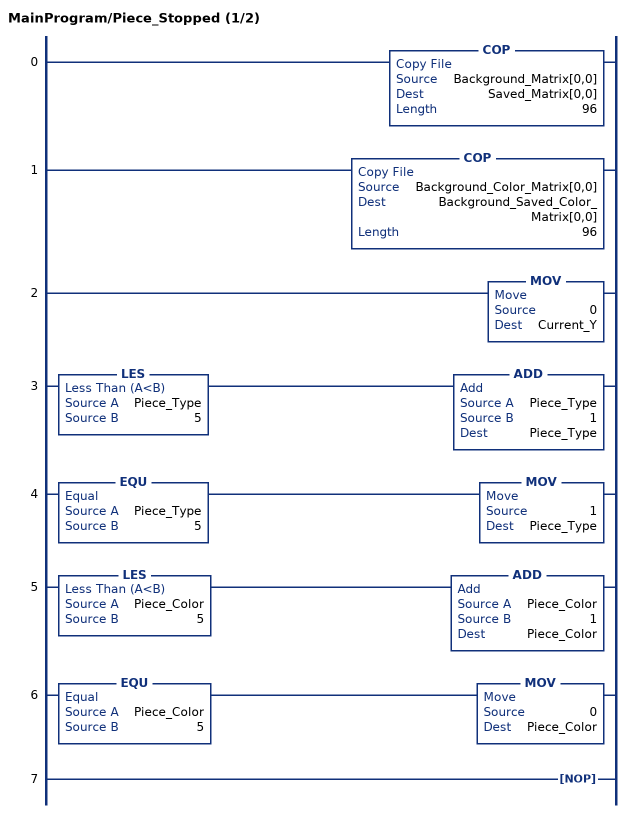
   0: COP(Background_Matrix[0,0],Saved_Matrix[0,0],96);
   1: COP(Background_Color_Matrix[0,0],Background_Saved_Color_Matrix[0,0],96);
   2: MOV(0,Current_Y);
   3: LES(Piece_Type,5)ADD(Piece_Type,1,Piece_Type);
   4: EQU(Piece_Type,5)MOV(1,Piece_Type);
   5: LES(Piece_Color,5)ADD(Piece_Color,1,Piece_Color);
   6: EQU(Piece_Color,5)MOV(0,Piece_Color);
   7: NOP();
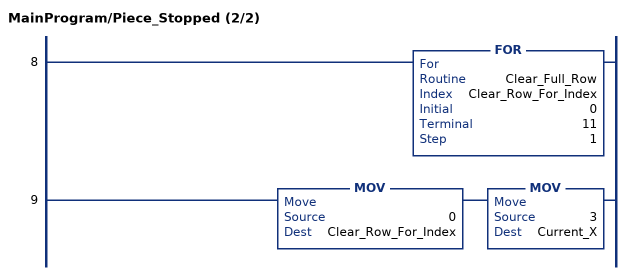
   8: FOR(Clear_Full_Row,Clear_Row_For_Index,0,11,1);
   9: MOV(0,Clear_Row_For_Index)MOV(3,Current_X);
END_ROUTINE

ROUTINE Update_Color_Matrix   (* ladder *)
END_ROUTINE

ROUTINE Update_Movement   (* ladder *)
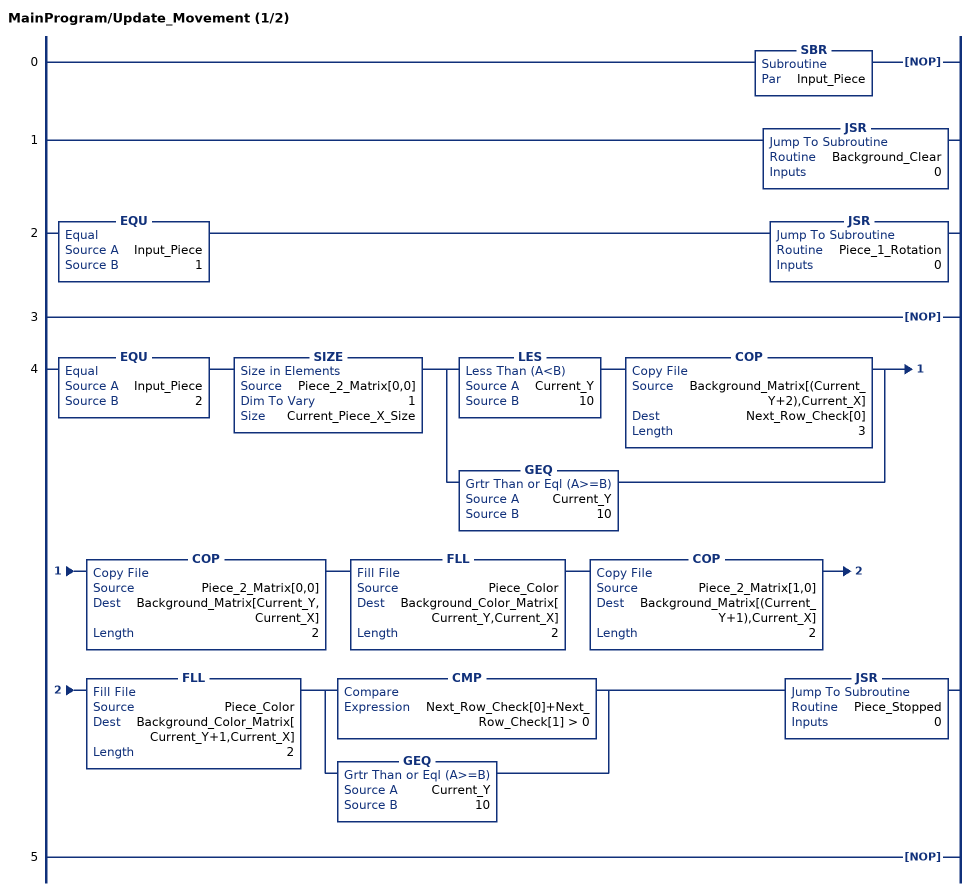
   0: SBR(Input_Piece)NOP();
   1: JSR(Background_Clear,0);
   2: EQU(Input_Piece,1)JSR(Piece_1_Rotation,0);
   3: NOP();
   4: EQU(Input_Piece,2)SIZE(Piece_2_Matrix[0,0],1,Current_Piece_X_Size)[LES(Current_Y,10) COP(Background_Matrix[(Current_Y+2),Current_X],Next_Row_Check[0],3) ,GEQ(Current_Y,10) ]COP(Piece_2_Matrix[0,0],Background_Matrix[Current_Y,Current_X],2)FLL(Piece_Color,Background_Color_Matrix[Current_Y,Current_X],2)COP(Piece_2_Matrix[1,0],Background_Matrix[(Current_Y+1),Current_X],2)FLL(Piece_Color,Background_Color_Matrix[Current_Y+1,Current_X],2)[CMP(Next_Row_Check[0]+Next_Row_Check[1] > 0) ,GEQ(Current_Y,10) ]JSR(Piece_Stopped,0);
   5: NOP();
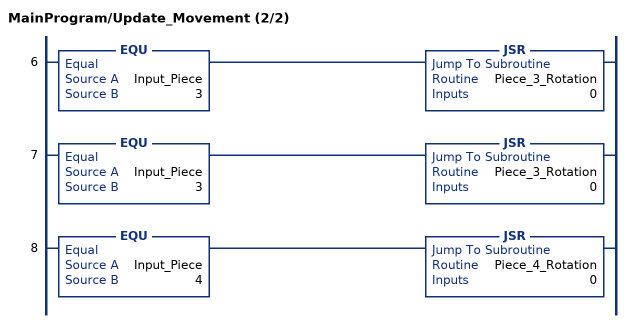
   6: EQU(Input_Piece,3)JSR(Piece_3_Rotation,0);
   7: EQU(Input_Piece,3)JSR(Piece_3_Rotation,0);
   8: EQU(Input_Piece,4)JSR(Piece_4_Rotation,0);
END_ROUTINE
END_PROGRAM
